TYPE ST_PSU_Outputs :
STRUCT
	bDisableOutput	: BOOL ;
	bReset			: BOOL ;
END_STRUCT
END_TYPE

(* stored: Version 1.1.0.1
   DUT ST_PSU_Outputs: Id {83720c42-48b4-4715-9bdb-3f3b194d5173} *)
